// TIA Portal V20 export
DATA_BLOCK "TEST"   // DB209
// stored: MemoryReserve 100, Namespace Unit1.Em4
   VAR RETAIN
      Bit : Array[0..99] of Bool;
      Dummy : Array[0..99] of Bool;
   END_VAR
BEGIN
   // Bit[0] : Vaccum Use
END_DATA_BLOCK
